// TIA Portal project "Automated_Warehouse-TIA_PORTAL_V17" (V17)
// Transport, store and retrieve boxes from a rack.

(* hardware
DEVICE "S7-1200 station_1"  S7-1200 Station
   slot 0: "Rack_0"  S7-1200 Rack  Rack  V1.0
   slot 1: "PLC_1"  CPU 1212C DC/DC/DC  6ES7 212-1AE40-0XB0  V4.5
*)

// ===== PLC "PLC_1"  CPU 1212C DC/DC/DC =====

VAR_GLOBAL   // PLC tag table "Default tag table"
   "Esteira de entrada" AT %Q0.0 : Bool;
   "Esteira de saida" AT %Q0.1 : Bool;
   "Esteira de carregamento" AT %Q0.2 : Bool;
   "Esteira de descarregamento" AT %Q0.3 : Bool;
   "Garfos de Entrada" AT %Q0.4 : Bool;
   "Garfos de Saida" AT %Q0.5 : Bool;
   "Elevador" AT %Q0.6 : Bool;
   "Led Verde" AT %Q0.7 : Bool;
   "Led Amarelo" AT %Q1.0 : Bool;
   "Led Vermelho" AT %Q1.1 : Bool;
   "Posicionador" AT %QD30 : DInt;
   "emergencia" AT %I0.0 : Bool;
   "botao start" AT %I0.1 : Bool;
   "botao stop" AT %I0.2 : Bool;
   "botao reset" AT %I0.3 : Bool;
   "Manual" AT %I0.4 : Bool;
   "Automático" AT %I0.5 : Bool;
   "sensor de entrada" AT %I0.6 : Bool;
   "sensor de carga" AT %I0.7 : Bool;
   "sensor garfo entrada" AT %I1.0 : Bool;
   "sensor eixo z" AT %I1.1 : Bool;
   "sensor garfo centralizado" AT %I1.2 : Bool;
   "sensor eixo x" AT %I1.3 : Bool;
   "sensor garfo saida" AT %I1.4 : Bool;
   "System_Byte" AT %MB1 : Byte;
   "FirstScan" AT %M1.0 : Bool;
   "DiagStatusUpdate" AT %M1.1 : Bool;
   "AlwaysTRUE" AT %M1.2 : Bool;
   "AlwaysFALSE" AT %M1.3 : Bool;
   "Clock_Byte" AT %MB0 : Byte;
   "Clock_10Hz" AT %M0.0 : Bool;
   "Clock_5Hz" AT %M0.1 : Bool;
   "Clock_2.5Hz" AT %M0.2 : Bool;
   "Clock_2Hz" AT %M0.3 : Bool;
   "Clock_1.25Hz" AT %M0.4 : Bool;
   "Clock_1Hz" AT %M0.5 : Bool;
   "Clock_0.625Hz" AT %M0.6 : Bool;
   "Clock_0.5Hz" AT %M0.7 : Bool;
END_VAR

DATA_BLOCK "DB"   // DB1
{ S7_Optimized_Access := 'TRUE' }
VERSION : 0.1
   VAR
      "M" : Array[0..15] of Bool;
      Habilita : Bool;
      Auto : Bool;
      Inicio : Bool;
      cont : Int;
      full : Bool;
      ciclo : Bool;
   END_VAR
BEGIN
END_DATA_BLOCK

// folder: System blocks/Program resources

DATA_BLOCK "Timer 0"   // DB2
{ S7_Optimized_Access := 'TRUE' }
AUTHOR : Simatic
FAMILY : IEC
NAME : IEC_TMR
VERSION : 1.0
// stored: InstanceOfName IEC_TIMER
"IEC_TIMER"
BEGIN
END_DATA_BLOCK

DATA_BLOCK "Timer 1"   // DB3
{ S7_Optimized_Access := 'TRUE' }
AUTHOR : Simatic
FAMILY : IEC
NAME : IEC_TMR
VERSION : 1.0
// stored: InstanceOfName IEC_TIMER
"IEC_TIMER"
BEGIN
END_DATA_BLOCK

DATA_BLOCK "Timer 2"   // DB4
{ S7_Optimized_Access := 'TRUE' }
AUTHOR : Simatic
FAMILY : IEC
NAME : IEC_TMR
VERSION : 1.0
// stored: InstanceOfName IEC_TIMER
"IEC_TIMER"
BEGIN
END_DATA_BLOCK

DATA_BLOCK "Timer 3"   // DB5
{ S7_Optimized_Access := 'TRUE' }
AUTHOR : Simatic
FAMILY : IEC
NAME : IEC_TMR
VERSION : 1.0
// stored: InstanceOfName IEC_TIMER
"IEC_TIMER"
BEGIN
END_DATA_BLOCK

DATA_BLOCK "Timer 4"   // DB6
{ S7_Optimized_Access := 'TRUE' }
AUTHOR : Simatic
FAMILY : IEC
NAME : IEC_TMR
VERSION : 1.0
// stored: InstanceOfName IEC_TIMER
"IEC_TIMER"
BEGIN
END_DATA_BLOCK

DATA_BLOCK "Timer 5"   // DB7
{ S7_Optimized_Access := 'TRUE' }
AUTHOR : Simatic
FAMILY : IEC
NAME : IEC_TMR
VERSION : 1.0
// stored: InstanceOfName IEC_TIMER
"IEC_TIMER"
BEGIN
END_DATA_BLOCK

DATA_BLOCK "Timer 6"   // DB8
{ S7_Optimized_Access := 'TRUE' }
AUTHOR : Simatic
FAMILY : IEC
NAME : IEC_TMR
VERSION : 1.0
// stored: InstanceOfName IEC_TIMER
"IEC_TIMER"
BEGIN
END_DATA_BLOCK

DATA_BLOCK "Timer 7"   // DB9
{ S7_Optimized_Access := 'TRUE' }
AUTHOR : Simatic
FAMILY : IEC
NAME : IEC_TMR
VERSION : 1.0
// stored: InstanceOfName IEC_TIMER
"IEC_TIMER"
BEGIN
END_DATA_BLOCK

DATA_BLOCK "Timer 8"   // DB10
{ S7_Optimized_Access := 'TRUE' }
AUTHOR : Simatic
FAMILY : IEC
NAME : IEC_TMR
VERSION : 1.0
// stored: InstanceOfName IEC_TIMER
"IEC_TIMER"
BEGIN
END_DATA_BLOCK

// folder: (top level)

FUNCTION "Block_1" : Void   // FC1, LAD
{ S7_Optimized_Access := 'TRUE' }
VERSION : 0.1
// Observação geral: o DB habilita serve para que eu possa apertar a qualquer momento o botao de desliga que o progama ja não avança para o passo seguinte.
   VAR_TEMP   // added for the SCL form of the ladder/FBD networks
      _w1 : Bool;
      _w2 : Bool;
   END_VAR
BEGIN

REGION Network 1: Lógica de Emergência
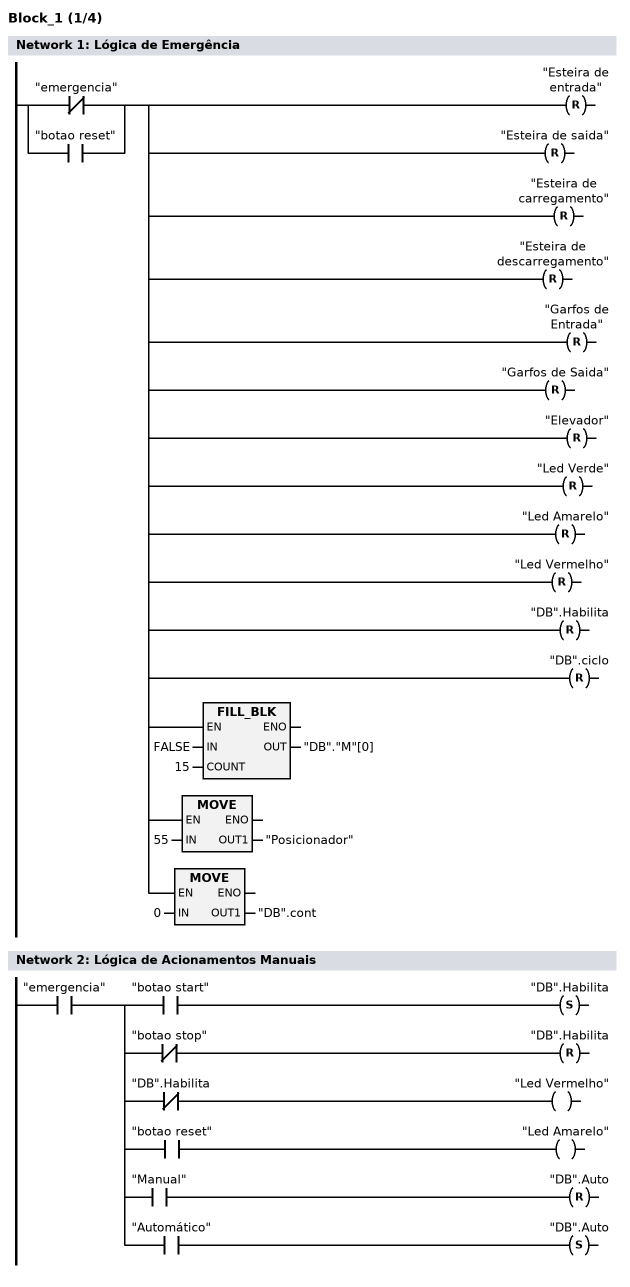
   RUNG wire#powerrail
      I_Contact( "emergencia" )
      wire#w1
      R_Coil( "Esteira de entrada" )
   END_RUNG
   RUNG wire#powerrail
      Contact( "botao reset" )
   END_RUNG wire#w1
   RUNG wire#w1
      R_Coil( "Esteira de saida" )
   END_RUNG
   RUNG wire#w1
      R_Coil( "Esteira de carregamento" )
   END_RUNG
   RUNG wire#w1
      R_Coil( "Esteira de descarregamento" )
   END_RUNG
   RUNG wire#w1
      R_Coil( "Garfos de Entrada" )
   END_RUNG
   RUNG wire#w1
      R_Coil( "Garfos de Saida" )
   END_RUNG
   RUNG wire#w1
      R_Coil( "Elevador" )
   END_RUNG
   RUNG wire#w1
      R_Coil( "Led Verde" )
   END_RUNG
   RUNG wire#w1
      R_Coil( "Led Amarelo" )
   END_RUNG
   RUNG wire#w1
      R_Coil( "Led Vermelho" )
   END_RUNG
   RUNG wire#w1
      R_Coil( "DB".Habilita )
   END_RUNG
   RUNG wire#w1
      R_Coil( "DB".ciclo )
   END_RUNG
   RUNG wire#w1
      FillBlockI(in := FALSE, count := 15, out => "DB"."M"[0])
   END_RUNG
   RUNG wire#w1
      Move(in := 55, out1 => "Posicionador")
   END_RUNG
   RUNG wire#w1
      Move(in := 0, out1 => "DB".cont)
   END_RUNG
   // the same network as SCL:
   IF NOT "emergencia" OR "botao reset" THEN
       "Esteira de entrada" := FALSE;
       "Esteira de saida" := FALSE;
       "Esteira de carregamento" := FALSE;
       "Esteira de descarregamento" := FALSE;
       "Garfos de Entrada" := FALSE;
       "Garfos de Saida" := FALSE;
       "Elevador" := FALSE;
       "Led Verde" := FALSE;
       "Led Amarelo" := FALSE;
       "Led Vermelho" := FALSE;
       "DB".Habilita := FALSE;
       "DB".ciclo := FALSE;
   END_IF;
   #_w1 := NOT "emergencia" OR "botao reset";
   IF #_w1 THEN
       FILL_BLK(IN := FALSE, COUNT := 15, OUT => "DB"."M"[0]);
       "Posicionador" := 55;
       "DB".cont := 0;
   END_IF;
END_REGION

REGION Network 2: Lógica de Acionamentos Manuais
   RUNG wire#powerrail
      Contact( "emergencia" )
      wire#w1
      Contact( "botao start" )
      S_Coil( "DB".Habilita )
   END_RUNG
   RUNG wire#w1
      I_Contact( "botao stop" )
      R_Coil( "DB".Habilita )
   END_RUNG
   RUNG wire#w1
      I_Contact( "DB".Habilita )
      Coil( "Led Vermelho" )
   END_RUNG
   RUNG wire#w1
      Contact( "botao reset" )
      Coil( "Led Amarelo" )
   END_RUNG
   RUNG wire#w1
      Contact( "Manual" )
      R_Coil( "DB".Auto )
   END_RUNG
   RUNG wire#w1
      Contact( "Automático" )
      S_Coil( "DB".Auto )
   END_RUNG
   // the same network as SCL:
   IF "emergencia" AND "botao start" THEN "DB".Habilita := TRUE; END_IF;
   IF "emergencia" AND NOT "botao stop" THEN "DB".Habilita := FALSE; END_IF;
   "Led Vermelho" := "emergencia" AND NOT "DB".Habilita;
   "Led Amarelo" := "emergencia" AND "botao reset";
   IF "emergencia" AND "Manual" THEN "DB".Auto := FALSE; END_IF;
   IF "emergencia" AND "Automático" THEN "DB".Auto := TRUE; END_IF;
END_REGION

REGION Network 3: Lógica do Processo (Modo Automático)
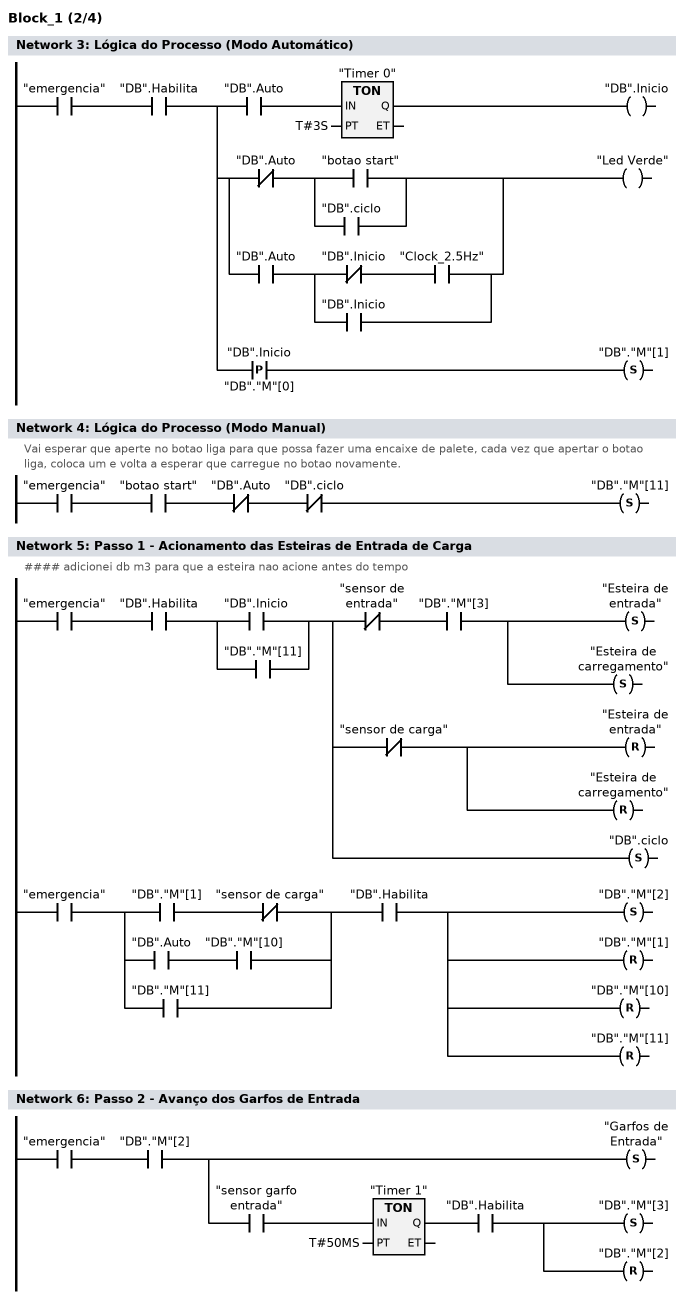
   #_w1 := "emergencia" AND "DB".Habilita;
   "Timer 0".TON(IN := #_w1 AND "DB".Auto, PT := T#3S);
   "DB".Inicio := "Timer 0".Q;
   "Led Verde" := #_w1 AND ((NOT "DB".Auto AND ("botao start" OR "DB".ciclo)) OR ("DB".Auto AND ((NOT "DB".Inicio AND "Clock_2.5Hz") OR "DB".Inicio)));
   #_w2 := #_w1 AND "DB".Inicio AND NOT "DB"."M"[0];   // rising edge of "DB".Inicio
   "DB"."M"[0] := "DB".Inicio;
   IF #_w2 THEN "DB"."M"[1] := TRUE; END_IF;
END_REGION

REGION Network 4: Lógica do Processo (Modo Manual)
   // Vai esperar que aperte no botao liga para que possa fazer uma encaixe de palete, cada vez que apertar o botao liga, coloca um e volta a esperar que carregue no botao novamente.
   RUNG wire#powerrail
      Contact( "emergencia" )
      Contact( "botao start" )
      I_Contact( "DB".Auto )
      I_Contact( "DB".ciclo )
      S_Coil( "DB"."M"[11] )
   END_RUNG
   // the same network as SCL:
   IF "emergencia" AND "botao start" AND NOT "DB".Auto AND NOT "DB".ciclo THEN "DB"."M"[11] := TRUE; END_IF;
END_REGION

REGION Network 5: Passo 1 - Acionamento das Esteiras de Entrada de Carga
   // #### adicionei db m3 para que a esteira nao acione antes do tempo
   RUNG wire#powerrail
      Contact( "emergencia" )
      Contact( "DB".Habilita )
      wire#w1
      Contact( "DB".Inicio )
      wire#w2
      I_Contact( "sensor de entrada" )
      Contact( "DB"."M"[3] )
      wire#w3
      S_Coil( "Esteira de entrada" )
   END_RUNG
   RUNG wire#w1
      Contact( "DB"."M"[11] )
   END_RUNG wire#w2
   RUNG wire#w3
      S_Coil( "Esteira de carregamento" )
   END_RUNG
   RUNG wire#w2
      I_Contact( "sensor de carga" )
      wire#w4
      R_Coil( "Esteira de entrada" )
   END_RUNG
   RUNG wire#w4
      R_Coil( "Esteira de carregamento" )
   END_RUNG
   RUNG wire#w2
      S_Coil( "DB".ciclo )
   END_RUNG
   RUNG wire#powerrail
      Contact( "emergencia" )
      wire#w5
      Contact( "DB"."M"[1] )
      I_Contact( "sensor de carga" )
      wire#w6
      Contact( "DB".Habilita )
      wire#w7
      S_Coil( "DB"."M"[2] )
   END_RUNG
   RUNG wire#w5
      Contact( "DB".Auto )
      Contact( "DB"."M"[10] )
   END_RUNG wire#w6
   RUNG wire#w5
      Contact( "DB"."M"[11] )
   END_RUNG wire#w6
   RUNG wire#w7
      R_Coil( "DB"."M"[1] )
   END_RUNG
   RUNG wire#w7
      R_Coil( "DB"."M"[10] )
   END_RUNG
   RUNG wire#w7
      R_Coil( "DB"."M"[11] )
   END_RUNG
   // the same network as SCL:
   #_w1 := "emergencia" AND "DB".Habilita AND ("DB".Inicio OR "DB"."M"[11]);
   IF #_w1 AND NOT "sensor de entrada" AND "DB"."M"[3] THEN
       "Esteira de entrada" := TRUE;
       "Esteira de carregamento" := TRUE;
   END_IF;
   IF #_w1 AND NOT "sensor de carga" THEN
       "Esteira de entrada" := FALSE;
       "Esteira de carregamento" := FALSE;
   END_IF;
   IF #_w1 THEN "DB".ciclo := TRUE; END_IF;
   #_w2 := "emergencia" AND (("DB"."M"[1] AND NOT "sensor de carga") OR ("DB".Auto AND "DB"."M"[10]) OR "DB"."M"[11]) AND "DB".Habilita;
   IF #_w2 THEN
       "DB"."M"[2] := TRUE;
       "DB"."M"[1] := FALSE;
       "DB"."M"[10] := FALSE;
       "DB"."M"[11] := FALSE;
   END_IF;
END_REGION

REGION Network 6: Passo 2 - Avanço dos Garfos de Entrada
   #_w1 := "emergencia" AND "DB"."M"[2];
   IF #_w1 THEN "Garfos de Entrada" := TRUE; END_IF;
   "Timer 1".TON(IN := #_w1 AND "sensor garfo entrada", PT := T#50MS);
   IF "Timer 1".Q AND "DB".Habilita THEN
       "DB"."M"[3] := TRUE;
       "DB"."M"[2] := FALSE;
   END_IF;
END_REGION

REGION Network 7: Passo 3 - Avanço do Elevador
   // ton para garantir que o elevador chegou pois o sensor eixo z somente atua quando estar em movimento 
   //  -> garantir que somente vá para o passo seguinte quando estiver ok
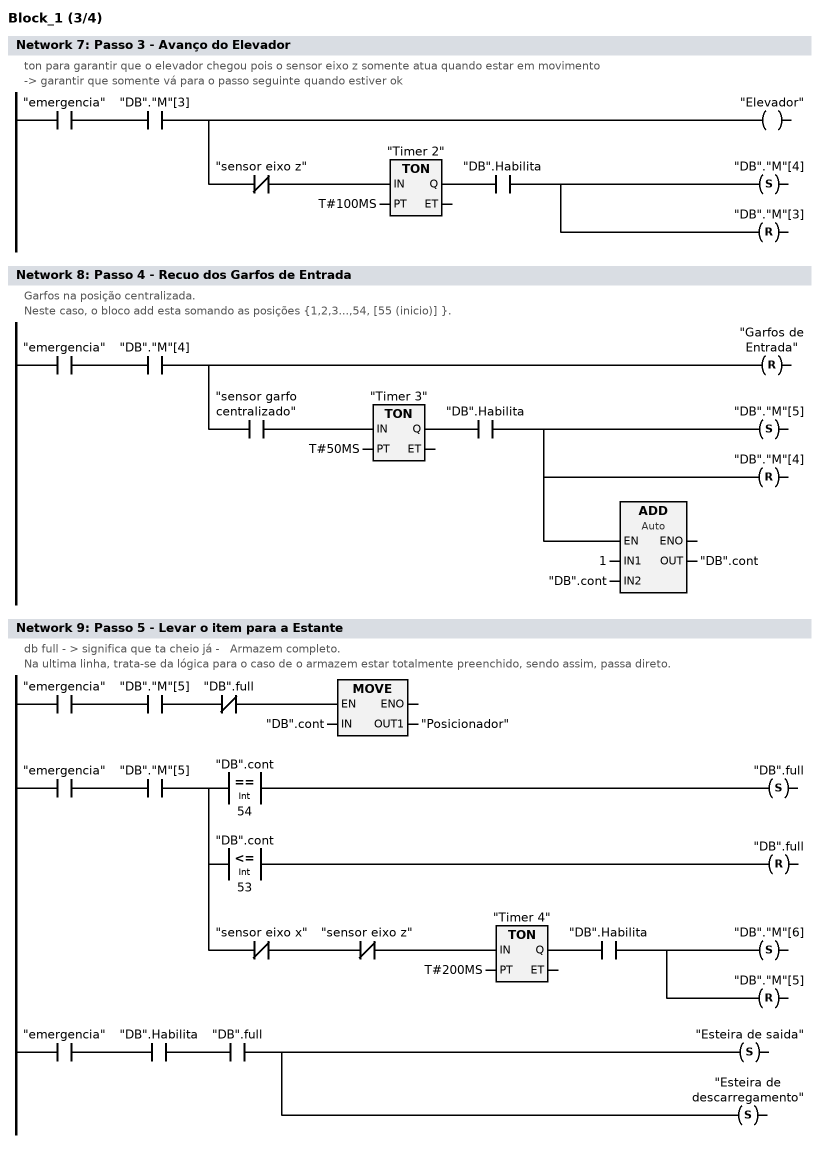
   "Elevador" := "emergencia" AND "DB"."M"[3];
   "Timer 2".TON(IN := "Elevador" AND NOT "sensor eixo z", PT := T#100MS);
   IF "Timer 2".Q AND "DB".Habilita THEN
       "DB"."M"[4] := TRUE;
       "DB"."M"[3] := FALSE;
   END_IF;
END_REGION

REGION Network 8: Passo 4 - Recuo dos Garfos de Entrada
   // Garfos na posição centralizada.
   // 
   // Neste caso, o bloco add esta somando as posições {1,2,3...,54, [55 (inicio)] }.
   #_w1 := "emergencia" AND "DB"."M"[4];
   IF #_w1 THEN "Garfos de Entrada" := FALSE; END_IF;
   "Timer 3".TON(IN := #_w1 AND "sensor garfo centralizado", PT := T#50MS);
   IF "Timer 3".Q AND "DB".Habilita THEN
       "DB"."M"[5] := TRUE;
       "DB"."M"[4] := FALSE;
       "DB".cont := 1 + "DB".cont;
   END_IF;
END_REGION

REGION Network 9: Passo 5 - Levar o item para a Estante
   // db full - > significa que ta cheio já -   Armazem completo.
   // 
   // Na ultima linha, trata-se da lógica para o caso de o armazem estar totalmente preenchido, sendo assim, passa direto.
   IF "emergencia" AND "DB"."M"[5] AND NOT "DB".full THEN "Posicionador" := "DB".cont; END_IF;
   #_w1 := "emergencia" AND "DB"."M"[5];
   IF #_w1 AND ("DB".cont = 54) THEN "DB".full := TRUE; END_IF;
   IF #_w1 AND ("DB".cont <= 53) THEN "DB".full := FALSE; END_IF;
   "Timer 4".TON(IN := #_w1 AND NOT "sensor eixo x" AND NOT "sensor eixo z", PT := T#200MS);
   IF "Timer 4".Q AND "DB".Habilita THEN
       "DB"."M"[6] := TRUE;
       "DB"."M"[5] := FALSE;
   END_IF;
   IF "emergencia" AND "DB".Habilita AND "DB".full THEN
       "Esteira de saida" := TRUE;
       "Esteira de descarregamento" := TRUE;
   END_IF;
END_REGION

REGION Network 10: Passo 6 - Avanço dos Garfos de Saida
   // Poscissiona o palete na estante. 
   // coloca (avança o palete )
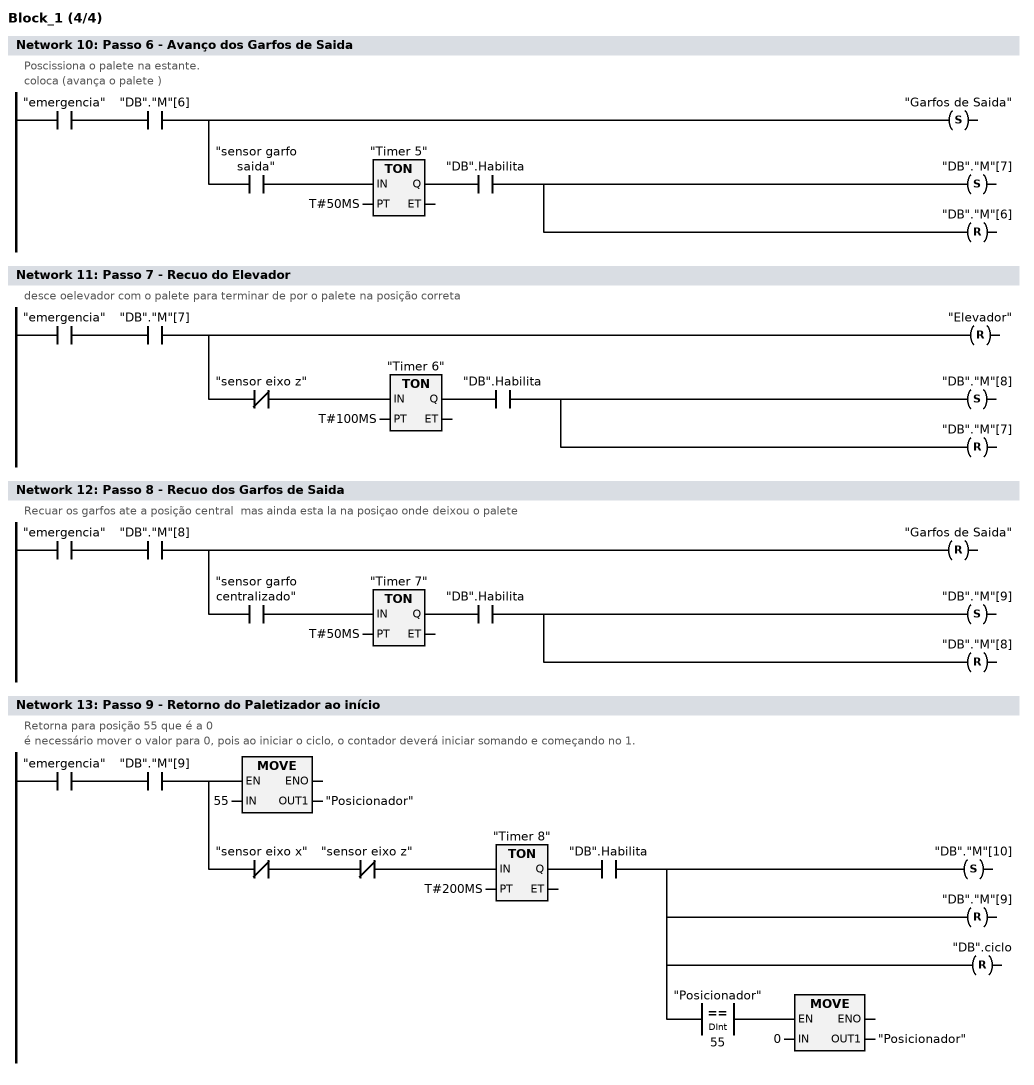
   #_w1 := "emergencia" AND "DB"."M"[6];
   IF #_w1 THEN "Garfos de Saida" := TRUE; END_IF;
   "Timer 5".TON(IN := #_w1 AND "sensor garfo saida", PT := T#50MS);
   IF "Timer 5".Q AND "DB".Habilita THEN
       "DB"."M"[7] := TRUE;
       "DB"."M"[6] := FALSE;
   END_IF;
END_REGION

REGION Network 11: Passo 7 - Recuo do Elevador
   // desce oelevador com o palete para terminar de por o palete na posição correta
   #_w1 := "emergencia" AND "DB"."M"[7];
   IF #_w1 THEN "Elevador" := FALSE; END_IF;
   "Timer 6".TON(IN := #_w1 AND NOT "sensor eixo z", PT := T#100MS);
   IF "Timer 6".Q AND "DB".Habilita THEN
       "DB"."M"[8] := TRUE;
       "DB"."M"[7] := FALSE;
   END_IF;
END_REGION

REGION Network 12: Passo 8 - Recuo dos Garfos de Saida
   // Recuar os garfos ate a posição central  mas ainda esta la na posiçao onde deixou o palete
   #_w1 := "emergencia" AND "DB"."M"[8];
   IF #_w1 THEN "Garfos de Saida" := FALSE; END_IF;
   "Timer 7".TON(IN := #_w1 AND "sensor garfo centralizado", PT := T#50MS);
   IF "Timer 7".Q AND "DB".Habilita THEN
       "DB"."M"[9] := TRUE;
       "DB"."M"[8] := FALSE;
   END_IF;
END_REGION

REGION Network 13: Passo 9 - Retorno do Paletizador ao início
   // Retorna para posição 55 que é a 0
   // é necessário mover o valor para 0, pois ao iniciar o ciclo, o contador deverá iniciar somando e começando no 1.
   #_w1 := "emergencia" AND "DB"."M"[9];
   IF #_w1 THEN "Posicionador" := 55; END_IF;
   "Timer 8".TON(IN := #_w1 AND NOT "sensor eixo x" AND NOT "sensor eixo z", PT := T#200MS);
   #_w2 := "Timer 8".Q AND "DB".Habilita;
   IF #_w2 THEN
       "DB"."M"[10] := TRUE;
       "DB"."M"[9] := FALSE;
       "DB".ciclo := FALSE;
   END_IF;
   IF #_w2 AND ("Posicionador" = 55) THEN "Posicionador" := 0; END_IF;
END_REGION
END_FUNCTION

FUNCTION "MHJ-PLC-Lab-Function-S71200" : Void   // FC9000, SCL
{ S7_Optimized_Access := 'TRUE' }
VERSION : 0.1
   VAR_TEMP
      rdTimeReturn : Int;
      outputTime : DTL;
      SyncVal : Byte;
      forVal : Int;
      forVal_2 : Int;
      Value : Byte;
   END_VAR
   VAR CONSTANT
      CompVal : Byte := 16#34;
      Value_01 : Byte := 16#11;
      Value_01_DW : DWord := 16#A165_D992;
      Value_02_DW : DWord := 16#58BE_4401;
   END_VAR
BEGIN

   #Value:=PEEK(area := 16#82,
        dbNumber := 0,
        byteOffset := 511);
   #Value := #Value + 1;

   POKE(area := 16#82,
        dbNumber := 0,
        byteOffset := 511,
        value := #Value);

   POKE(area:=16#81,
        dbNumber:=0,
        byteOffset:=1016,
        value:=#Value_01_DW);
   POKE(area := 16#81,
        dbNumber := 0,
        byteOffset := 1020,
        value := #Value_02_DW);

   POKE(area := 16#81,
        dbNumber := 0,
        byteOffset := 511,
        value := B#16#00);

   FOR #forVal := 0 TO 120 DO
       FOR #forVal_2:=0 TO 10 DO
           #rdTimeReturn:=RD_SYS_T(#outputTime);
           #rdTimeReturn := WR_SYS_T(#outputTime);
           #rdTimeReturn := RD_SYS_T(#outputTime);
           #rdTimeReturn := WR_SYS_T(#outputTime);
       END_FOR;
       #SyncVal:= PEEK(area := 16#81,
                      dbNumber := 0,
                      byteOffset := 511);
       IF #SyncVal = #CompVal THEN
          GOTO M_1;
       END_IF;
   END_FOR;
   RETURN;

   M_1:
   POKE(area := 16#81,
        dbNumber := 0,
        byteOffset := 511,
        value := B#16#0);
END_FUNCTION

ORGANIZATION_BLOCK "Main"   // OB1, LAD, ProgramCycle
TITLE = "Main Program Sweep (Cycle)"
{ S7_Optimized_Access := 'TRUE' }
VERSION : 0.1
   VAR_INPUT
      Initial_Call : Bool;   // Initial call of this OB
      Remanence : Bool;   // =True, if remanent data are available
   END_VAR
BEGIN

REGION Network 1
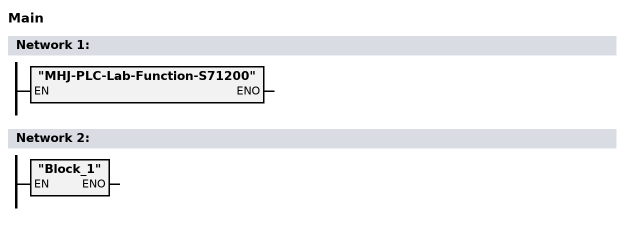
   RUNG wire#powerrail
      "MHJ-PLC-Lab-Function-S71200"()
   END_RUNG
   // the same network as SCL:
   "MHJ-PLC-Lab-Function-S71200"();
END_REGION

REGION Network 2
   RUNG wire#powerrail
      "Block_1"()
   END_RUNG
   // the same network as SCL:
   "Block_1"();
END_REGION
END_ORGANIZATION_BLOCK